(* PLC project  *)

PROGRAM OB1

(* FBD diagram, written out as Structured Text *)
END_PROGRAM

FUNCTION_BLOCK FB_Monitor

            TRUE
          
END_FUNCTION_BLOCK

PROGRAM OB100

            FALSE
          
END_PROGRAM
